# EPICS autosave request: softGlueApp/Db/gate_settings.req
$(P)$(H)$(GATE)_IN1_Signal
$(P)$(H)$(GATE)_IN2_Signal
$(P)$(H)$(GATE)_OUT_Signal
